FUNCTION_BLOCK Percentual
VAR_INPUT
	VAR_1:DINT;
	VAR_2:DINT;
END_VAR
VAR_OUTPUT
	OUTPUT:DINT;
END_VAR

//Retorna o valor percentual da variável 1 em relação a variável 2
OUTPUT := SEL(VAR_2 > 0, 0,(VAR_1*100/VAR_2*100)/100);

END_FUNCTION_BLOCK

(* stored: Version 1.1.0.1, ProductVersion 3.1.4024.14
   POU Percentual: Id {4dde3a47-103e-40dc-a643-55cc975f94e9}, SpecialFunc None *)
